// TIA Portal V20 export
FUNCTION_BLOCK "Diag"   // FB60, FBD
TITLE = diagnose
{ S7_Optimized_Access := 'TRUE' }
// stored: AutoNumber false, MemoryReserve 100, SetENOAutomatically false
   VAR
      Var { ExternalAccessible := 'False'; ExternalVisible := 'False'; ExternalWritable := 'False'} : "TypeVar";
      Plc { ExternalAccessible := 'False'; ExternalVisible := 'False'; ExternalWritable := 'False'} : "Diag_PLCCheck";
      PlcData { ExternalAccessible := 'False'; ExternalVisible := 'False'; ExternalWritable := 'False'} : "UserDiag_typePLC";   // PLC diagnostics data
      IoSys1 { ExternalAccessible := 'False'; ExternalVisible := 'False'; ExternalWritable := 'False'} : "Diag_IOSystemCheck";
      IoDataSys1 { ExternalAccessible := 'False'; ExternalVisible := 'False'; ExternalWritable := 'False'} : "UserDiag_typeIOSystem";   // IO-System diagnostics data
   END_VAR
BEGIN

REGION Network 1: Call startup and diagnostics of PLC
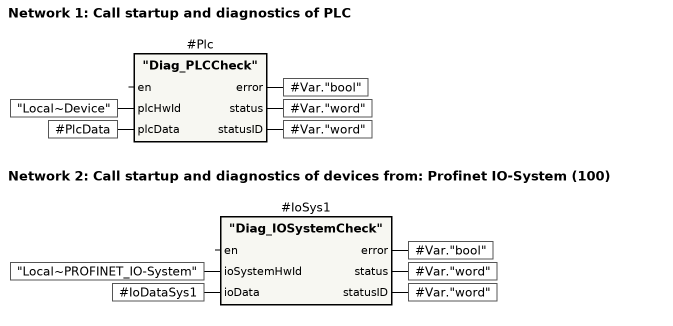
   #Plc(plcHwId := "Local~Device",   // "Diag_PLCCheck"
        plcData := #PlcData,
        error => #Var."bool",
        status => #Var."word",
        statusID => #Var."word");
END_REGION

REGION Network 2: Call startup and diagnostics of devices from: Profinet IO-System (100)
   #IoSys1(ioSystemHwId := "Local~PROFINET_IO-System",   // "Diag_IOSystemCheck"
           ioData := #IoDataSys1,
           error => #Var."bool",
           status => #Var."word",
           statusID => #Var."word");
END_REGION
END_FUNCTION_BLOCK
